PROGRAM EnOceanCom
VAR
	fbKL6581: FB_KL6581;
	fbEnOceanSearch: FB_EnOcean_Search;
END_VAR

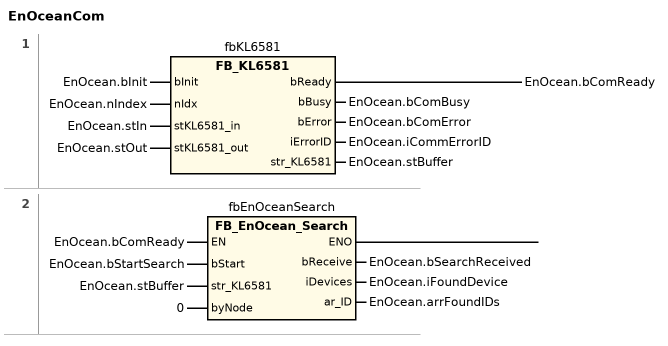
// NETWORK 1
fbKL6581(
    bInit := EnOcean.bInit,
    nIdx := EnOcean.nIndex,
    stKL6581_in := EnOcean.stIn,
    stKL6581_out := EnOcean.stOut,
    bBusy => EnOcean.bComBusy,
    bError => EnOcean.bComError,
    iErrorID => EnOcean.iCommErrorID,
    str_KL6581 => EnOcean.stBuffer); // FB_KL6581
EnOcean.bComReady := fbKL6581.bReady;

// NETWORK 2
IF EnOcean.bComReady THEN
    fbEnOceanSearch(
        bStart := EnOcean.bStartSearch,
        str_KL6581 := EnOcean.stBuffer,
        byNode := 0,
        bReceive => EnOcean.bSearchReceived,
        iDevices => EnOcean.iFoundDevice,
        ar_ID => EnOcean.arrFoundIDs); // FB_EnOcean_Search
END_IF

END_PROGRAM

(* stored: Version 1.1.0.1, ProductVersion 3.1.4024.11
   POU EnOceanCom: Id {cc9cc52e-3ed0-46d7-ad4f-471667a606b0}, SpecialFunc None *)
